// TIA Portal project "141db_PLcen hasera" (V15.1)

(* hardware
DEVICE "S7-1200 station_1"  S7-1200 Station
   slot 0: "Rack_0"  S7-1200 Rack  Rack  V1.0
   slot 1: "PLC_1"  CPU 1214C AC/DC/Rly  6ES7 214-1BG40-0XB0  V4.2
   slot 3: "AQ 1x12BIT_1"  AQ1 signal board  6ES7 232-4HA30-0XB0  V1.0
*)

// ===== PLC "PLC_1"  CPU 1214C AC/DC/Rly =====

VAR_GLOBAL   // PLC tag table "Tabla de variables estándar"
   "Etapa0" AT %M16.0 : Bool;
   "S1" AT %I1.0 : Bool;
   "CP" AT %I1.3 : Bool;
   "S2" AT %I1.1 : Bool;
   "P1" AT %Q1.0 : Bool;
   "S3" AT %I1.2 : Bool;
   "CG" AT %I1.4 : Bool;
   "Etapa1" AT %M16.1 : Bool;
   "Etapa2" AT %M16.2 : Bool;
   "Etapa3" AT %M16.3 : Bool;
   "Etapa4" AT %M16.4 : Bool;
   "Etapa5" AT %M16.5 : Bool;
   "Etapa6" AT %M16.6 : Bool;
   "P3" AT %Q1.2 : Bool;
   "P2" AT %Q1.1 : Bool;
END_VAR

// folder: System blocks/Program resources

DATA_BLOCK "Temporizador1"   // DB2
{ S7_Optimized_Access := 'TRUE' }
AUTHOR : Simatic
FAMILY : IEC
NAME : IEC_TMR
VERSION : 1.0
// stored: InstanceOfName IEC_TIMER
"IEC_TIMER"
BEGIN
END_DATA_BLOCK

DATA_BLOCK "Temporizador2"   // DB3
{ S7_Optimized_Access := 'TRUE' }
AUTHOR : Simatic
FAMILY : IEC
NAME : IEC_TMR
VERSION : 1.0
// stored: InstanceOfName IEC_TIMER
"IEC_TIMER"
BEGIN
END_DATA_BLOCK

DATA_BLOCK "Temporizador4"   // DB4
{ S7_Optimized_Access := 'TRUE' }
AUTHOR : Simatic
FAMILY : IEC
NAME : IEC_TMR
VERSION : 1.0
// stored: InstanceOfName IEC_TIMER
"IEC_TIMER"
BEGIN
END_DATA_BLOCK

// folder: (top level)

ORGANIZATION_BLOCK "Main"   // OB1, LAD, ProgramCycle
TITLE = "Main Program Sweep (Cycle)"
{ S7_Optimized_Access := 'TRUE' }
VERSION : 0.1
   VAR_INPUT
      Initial_Call : Bool;   // Initial call of this OB
      Remanence : Bool;   // =True, if remanent data are available
   END_VAR
BEGIN

REGION Network 1
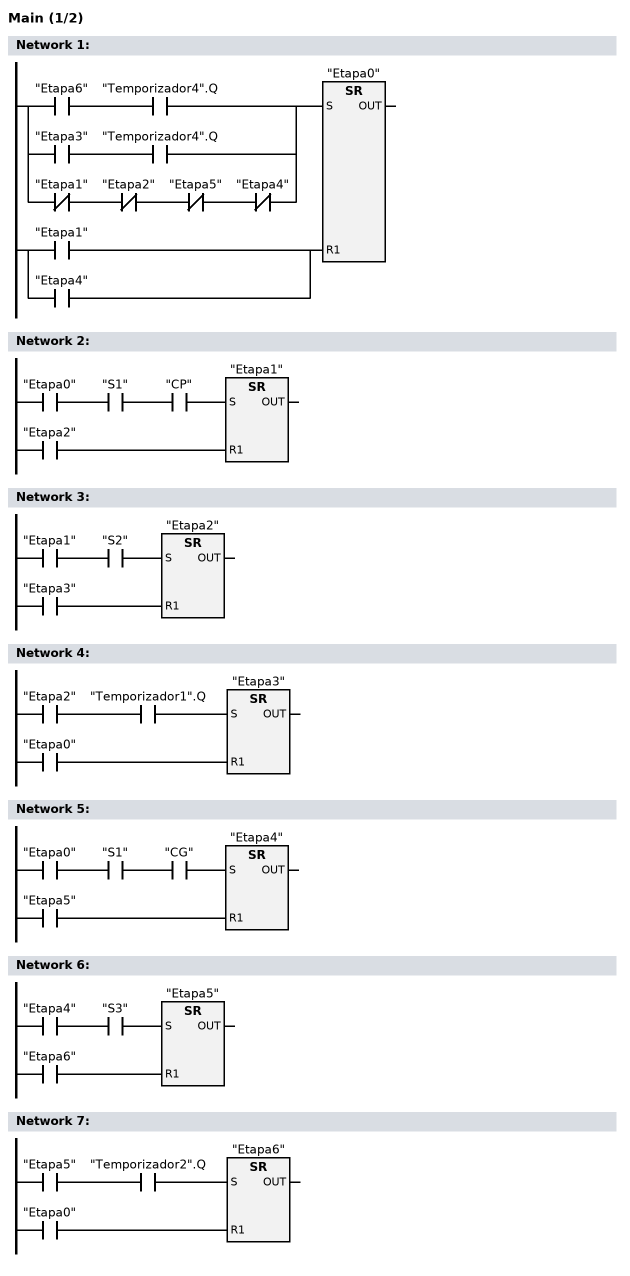
   RUNG wire#powerrail
      Contact( "Etapa6" )
      Contact( "Temporizador4".Q )
      wire#w1
      S_SR(operand := "Etapa0", r1 := wire#w2)
   END_RUNG
   RUNG wire#powerrail
      Contact( "Etapa3" )
      Contact( "Temporizador4".Q )
   END_RUNG wire#w1
   RUNG wire#powerrail
      I_Contact( "Etapa1" )
      I_Contact( "Etapa2" )
      I_Contact( "Etapa5" )
      I_Contact( "Etapa4" )
   END_RUNG wire#w1
   RUNG wire#powerrail
      Contact( "Etapa1" )
   END_RUNG wire#w2
   RUNG wire#powerrail
      Contact( "Etapa4" )
   END_RUNG wire#w2
   // the same network as SCL:
   IF ("Etapa6" AND "Temporizador4".Q) OR ("Etapa3" AND "Temporizador4".Q) OR (NOT "Etapa1" AND NOT "Etapa2" AND NOT "Etapa5" AND NOT "Etapa4") THEN
       "Etapa0" := TRUE;   // SR flip-flop
   END_IF;
   IF "Etapa1" OR "Etapa4" THEN "Etapa0" := FALSE; END_IF;
END_REGION

REGION Network 2
   RUNG wire#powerrail
      Contact( "Etapa0" )
      Contact( "S1" )
      Contact( "CP" )
      S_SR(operand := "Etapa1", r1 := wire#w1)
   END_RUNG
   RUNG wire#powerrail
      Contact( "Etapa2" )
   END_RUNG wire#w1
   // the same network as SCL:
   IF "Etapa0" AND "S1" AND "CP" THEN
       "Etapa1" := TRUE;   // SR flip-flop
   END_IF;
   IF "Etapa2" THEN "Etapa1" := FALSE; END_IF;
END_REGION

REGION Network 3
   RUNG wire#powerrail
      Contact( "Etapa1" )
      Contact( "S2" )
      S_SR(operand := "Etapa2", r1 := wire#w1)
   END_RUNG
   RUNG wire#powerrail
      Contact( "Etapa3" )
   END_RUNG wire#w1
   // the same network as SCL:
   IF "Etapa1" AND "S2" THEN
       "Etapa2" := TRUE;   // SR flip-flop
   END_IF;
   IF "Etapa3" THEN "Etapa2" := FALSE; END_IF;
END_REGION

REGION Network 4
   RUNG wire#powerrail
      Contact( "Etapa2" )
      Contact( "Temporizador1".Q )
      S_SR(operand := "Etapa3", r1 := wire#w1)
   END_RUNG
   RUNG wire#powerrail
      Contact( "Etapa0" )
   END_RUNG wire#w1
   // the same network as SCL:
   IF "Etapa2" AND "Temporizador1".Q THEN
       "Etapa3" := TRUE;   // SR flip-flop
   END_IF;
   IF "Etapa0" THEN "Etapa3" := FALSE; END_IF;
END_REGION

REGION Network 5
   RUNG wire#powerrail
      Contact( "Etapa0" )
      Contact( "S1" )
      Contact( "CG" )
      S_SR(operand := "Etapa4", r1 := wire#w1)
   END_RUNG
   RUNG wire#powerrail
      Contact( "Etapa5" )
   END_RUNG wire#w1
   // the same network as SCL:
   IF "Etapa0" AND "S1" AND "CG" THEN
       "Etapa4" := TRUE;   // SR flip-flop
   END_IF;
   IF "Etapa5" THEN "Etapa4" := FALSE; END_IF;
END_REGION

REGION Network 6
   RUNG wire#powerrail
      Contact( "Etapa4" )
      Contact( "S3" )
      S_SR(operand := "Etapa5", r1 := wire#w1)
   END_RUNG
   RUNG wire#powerrail
      Contact( "Etapa6" )
   END_RUNG wire#w1
   // the same network as SCL:
   IF "Etapa4" AND "S3" THEN
       "Etapa5" := TRUE;   // SR flip-flop
   END_IF;
   IF "Etapa6" THEN "Etapa5" := FALSE; END_IF;
END_REGION

REGION Network 7
   RUNG wire#powerrail
      Contact( "Etapa5" )
      Contact( "Temporizador2".Q )
      S_SR(operand := "Etapa6", r1 := wire#w1)
   END_RUNG
   RUNG wire#powerrail
      Contact( "Etapa0" )
   END_RUNG wire#w1
   // the same network as SCL:
   IF "Etapa5" AND "Temporizador2".Q THEN
       "Etapa6" := TRUE;   // SR flip-flop
   END_IF;
   IF "Etapa0" THEN "Etapa6" := FALSE; END_IF;
END_REGION

REGION Network 8
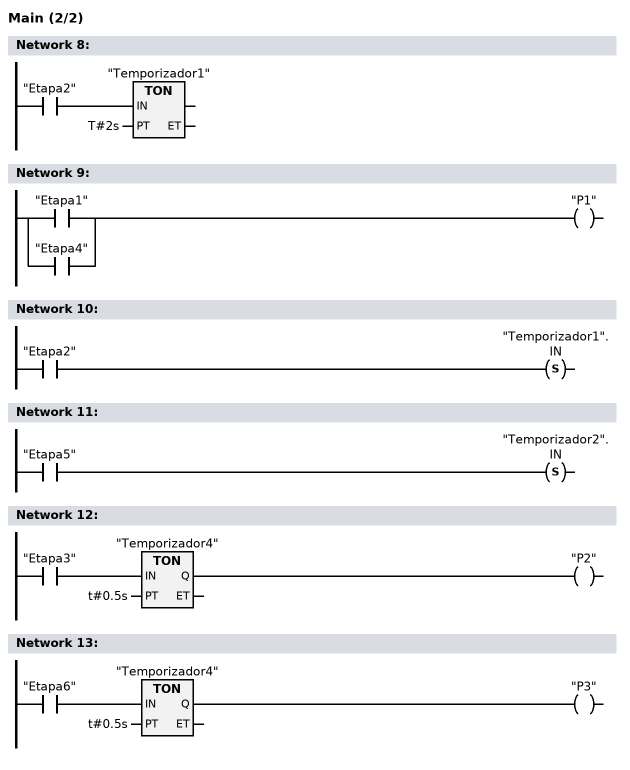
   "Temporizador1".TON(IN := "Etapa2", PT := T#2s);
END_REGION

REGION Network 9
   RUNG wire#powerrail
      Contact( "Etapa1" )
      wire#w1
      Coil( "P1" )
   END_RUNG
   RUNG wire#powerrail
      Contact( "Etapa4" )
   END_RUNG wire#w1
   // the same network as SCL:
   "P1" := "Etapa1" OR "Etapa4";
END_REGION

REGION Network 10
   RUNG wire#powerrail
      Contact( "Etapa2" )
      S_Coil( "Temporizador1".IN )
   END_RUNG
   // the same network as SCL:
   IF "Etapa2" THEN "Temporizador1".IN := TRUE; END_IF;
END_REGION

REGION Network 11
   RUNG wire#powerrail
      Contact( "Etapa5" )
      S_Coil( "Temporizador2".IN )
   END_RUNG
   // the same network as SCL:
   IF "Etapa5" THEN "Temporizador2".IN := TRUE; END_IF;
END_REGION

REGION Network 12
   "Temporizador4".TON(IN := "Etapa3", PT := t#0.5s);
   "P2" := "Temporizador4".Q;
END_REGION

REGION Network 13
   "Temporizador4".TON(IN := "Etapa6", PT := t#0.5s);
   "P3" := "Temporizador4".Q;
END_REGION
END_ORGANIZATION_BLOCK